TYPE arLiftAxis :
STRUCT
	lift : ARRAY[0..1] OF FB_remAxisMapping;
END_STRUCT
END_TYPE

(* stored: Version 1.1.0.1, ProductVersion 3.1.4024.12
   DUT arLiftAxis: Id {d7d57c75-bbdd-497d-9f25-c8ff05048bd0} *)
